        // ===========================================
        // STEP 350: MagnScanNGProcess
        // ===========================================
        STEP_ST10_Flow15_FRobot_3_MagnScanNGProcess:
            // No actions in XML

            // Transition to next step: 699
            IF TRUE THEN  // Sequential transition - review XML for actual condition
                #State := STEP_ST10_Flow15_FRobot_3_OKPutProcessFinish;
            END_IF;

        // ===========================================
        // STEP 699: OKPutProcessFinish
        // ===========================================
        STEP_ST10_Flow15_FRobot_3_OKPutProcessFinish:
            // Action Qualifier=S
            // Token: #ioPM_Inface.ProcessComplete
            #ioPM_Inface.ProcessComplete := TRUE;
            // Action Qualifier=R
            // Token: #ioPM_Inface.ProcessStart
            #ioPM_Inface.ProcessStart := FALSE;

            // Transition to next step: 355
            IF TRUE THEN  // Sequential transition - review XML for actual condition
                #State := STEP_ST10_Flow15_FRobot_3_StartRobotScanRing;
            END_IF;

        // ===========================================
        // STEP 355: StartRobotScanRing
        // ===========================================
        STEP_ST10_Flow15_FRobot_3_StartRobotScanRing:
            // Action Qualifier=N
            // Token: "KukaRobot3_CtrlDB".sPLCtoROB.User.Cycle.DI261_ScanRingReq
            "KukaRobot3_CtrlDB".sPLCtoROB.User.Cycle.DI261_ScanRingReq;

            // Transition to next step: 549
            IF TRUE THEN  // Sequential transition - review XML for actual condition
                #State := STEP_ST10_Flow15_FRobot_3_PressShaftPutProcessFinish;
            END_IF;

        // ===========================================
        // STEP 549: PressShaftPutProcessFinish
        // ===========================================
        STEP_ST10_Flow15_FRobot_3_PressShaftPutProcessFinish:
            // Action Qualifier=S
            // Token: #ioPM_Inface.ProcessComplete
            #ioPM_Inface.ProcessComplete := TRUE;
            // Action Qualifier=R
            // Token: #ioPM_Inface.ProcessStart
            #ioPM_Inface.ProcessStart := FALSE;

            // Transition to next step: 255
            IF TRUE THEN  // Sequential transition - review XML for actual condition
                #State := STEP_ST10_Flow15_FRobot_3_DataMove_1;
            END_IF;

        // ===========================================
        // STEP 255: DataMove_1
        // ===========================================
        STEP_ST10_Flow15_FRobot_3_DataMove_1:
            // Action Qualifier=N, Event="S1"
            // Token: "AutoProcessData".F_Robot3Grip2 := "AutoProcessData".C_MagnScanNGBuffer
            "AutoProcessData".F_Robot3Grip2 := "AutoProcessData".C_MagnScanNGBuffer;
            // Action Qualifier=N, Event="S1"
            // Token: "AutoProcessData".C_MagnScanNGBuffer := "AutoProcessData".ClearData
            "AutoProcessData".C_MagnScanNGBuffer := "AutoProcessData".ClearData;

            // Transition to next step: 382
            IF TRUE THEN  // Sequential transition - review XML for actual condition
                #State := STEP_ST10_Flow15_FRobot_3_Grip2SensorError;
            END_IF;

        // ===========================================
        // STEP 382: Grip2SensorError
        // ===========================================
        STEP_ST10_Flow15_FRobot_3_Grip2SensorError:
            // Action Qualifier=S
            // Token: "ST10_DeviceError".F.Robot_3.Grip2SensorCheckError
            "ST10_DeviceError".F.Robot_3.Grip2SensorCheckError := TRUE;

            // Transition to next step: 253
            IF TRUE THEN  // Sequential transition - review XML for actual condition
                #State := STEP_ST10_Flow15_FRobot_3_DataMove;
            END_IF;

        // ===========================================
        // STEP 253: DataMove
        // ===========================================
        STEP_ST10_Flow15_FRobot_3_DataMove:
            // Action Qualifier=N, Event="S1"
            // Token: "AutoProcessData".F_Robot3Grip1 := "AutoProcessData".C_GlueNGBuffer
            "AutoProcessData".F_Robot3Grip1 := "AutoProcessData".C_GlueNGBuffer;
            // Action Qualifier=N, Event="S1"
            // Token: "AutoProcessData".C_GlueNGBuffer := "AutoProcessData".ClearData
            "AutoProcessData".C_GlueNGBuffer := "AutoProcessData".ClearData;

            // Transition to next step: 919
            IF TRUE THEN  // Sequential transition - review XML for actual condition
                #State := STEP_ST10_Flow15_FRobot_3_MasteringTestFinish;
            END_IF;

        // ===========================================
        // STEP 919: MasteringTestFinish
        // ===========================================
        STEP_ST10_Flow15_FRobot_3_MasteringTestFinish:
            // Action Qualifier=R
            // Token: "Robot_DB".Robot_3.MasteringTest_Req
            "Robot_DB".Robot_3.MasteringTest_Req := FALSE;

            // Transition to next step: 900
            IF TRUE THEN  // Sequential transition - review XML for actual condition
                #State := STEP_ST10_Flow15_FRobot_3_S_900;
            END_IF;

        // ===========================================
        // STEP 900: 900
        // ===========================================
        STEP_ST10_Flow15_FRobot_3_S_900:
            // No actions in XML

            // Transition to next step: 309
            IF TRUE THEN  // Sequential transition - review XML for actual condition
                #State := STEP_ST10_Flow15_FRobot_3_WaitRobotReachPos1;
            END_IF;

        // ===========================================
        // STEP 309: WaitRobotReachPos1
        // ===========================================
        STEP_ST10_Flow15_FRobot_3_WaitRobotReachPos1:
            // No actions in XML

            // Transition to next step: 335
            IF TRUE THEN  // Sequential transition - review XML for actual condition
                #State := STEP_ST10_Flow15_FRobot_3_RobotScanGripperReachPos1;
            END_IF;

        // ===========================================
        // STEP 335: RobotScanGripperReachPos1
        // ===========================================
        STEP_ST10_Flow15_FRobot_3_RobotScanGripperReachPos1:
            // No actions in XML

            // Transition to next step: 267
            IF TRUE THEN  // Sequential transition - review XML for actual condition
                #State := STEP_ST10_Flow15_FRobot_3_Data_Clear_7;
            END_IF;

        // ===========================================
        // STEP 267: Data Clear_7
        // ===========================================
        STEP_ST10_Flow15_FRobot_3_Data_Clear_7:
            // Action Qualifier=N, Event="S1"
            // Token: "AutoProcessData".F_Robot3Grip1 := "AutoProcessData".ClearData
            "AutoProcessData".F_Robot3Grip1 := "AutoProcessData".ClearData;

            // Transition to next step: 705
            IF TRUE THEN  // Sequential transition - review XML for actual condition
                #State := STEP_ST10_Flow15_FRobot_3_WaitR1MaintenPosFinsh_1;
            END_IF;

        // ===========================================
        // STEP 705: WaitR1MaintenPosFinsh_1
        // ===========================================
        STEP_ST10_Flow15_FRobot_3_WaitR1MaintenPosFinsh_1:
            // Action Qualifier=R
            // Token: "AutoProcessControl".Robot_3.MaintenanceRequest
            "AutoProcessControl".Robot_3.MaintenanceRequest := FALSE;

            // Transition to next step: 500
            IF TRUE THEN  // Sequential transition - review XML for actual condition
                #State := STEP_ST10_Flow15_FRobot_3_PressShaftPutProcess;
            END_IF;

        // ===========================================
        // STEP 500: PressShaftPutProcess
        // ===========================================
        STEP_ST10_Flow15_FRobot_3_PressShaftPutProcess:
            // No actions in XML

            // Transition to next step: 376
            IF TRUE THEN  // Sequential transition - review XML for actual condition
                #State := STEP_ST10_Flow15_FRobot_3_StartRobotNG3Put;
            END_IF;

        // ===========================================
        // STEP 376: StartRobotNG3Put
        // ===========================================
        STEP_ST10_Flow15_FRobot_3_StartRobotNG3Put:
            // Action Qualifier=N
            // Token: "KukaRobot3_CtrlDB".sPLCtoROB.User.Cycle.DI267_LoadScanNGReq3
            "KukaRobot3_CtrlDB".sPLCtoROB.User.Cycle.DI267_LoadScanNGReq3;

            // Transition to next step: 333
            IF TRUE THEN  // Sequential transition - review XML for actual condition
                #State := STEP_ST10_Flow15_FRobot_3_RobotTaskSelect;
            END_IF;

        // ===========================================
        // STEP 333: RobotTaskSelect
        // ===========================================
        STEP_ST10_Flow15_FRobot_3_RobotTaskSelect:
            // No actions in XML

            // Transition to next step: 800
            IF TRUE THEN  // Sequential transition - review XML for actual condition
                #State := STEP_ST10_Flow15_FRobot_3_NG_3_PutProcess;
            END_IF;

        // ===========================================
        // STEP 800: NG 3 PutProcess
        // ===========================================
        STEP_ST10_Flow15_FRobot_3_NG_3_PutProcess:
            // No actions in XML

            // Transition to next step: 133
            IF TRUE THEN  // Sequential transition - review XML for actual condition
                #State := STEP_ST10_Flow15_FRobot_3_Brake_Test;
            END_IF;

        // ===========================================
        // STEP 133: Brake_Test
        // ===========================================
        STEP_ST10_Flow15_FRobot_3_Brake_Test:
            // Action Qualifier=R
            // Token: #ioPM_Inface.ProcessComplete
            #ioPM_Inface.ProcessComplete := FALSE;
            // Action Qualifier=S
            // Token: #ioPM_Inface.ProcessStart
            #ioPM_Inface.ProcessStart := TRUE;

            // Transition to next step: 365
            IF TRUE THEN  // Sequential transition - review XML for actual condition
                #State := STEP_ST10_Flow15_FRobot_3_WaitRobotFinish_7;
            END_IF;

        // ===========================================
        // STEP 365: WaitRobotFinish_7
        // ===========================================
        STEP_ST10_Flow15_FRobot_3_WaitRobotFinish_7:
            // No actions in XML

            // Transition to next step: 331
            IF TRUE THEN  // Sequential transition - review XML for actual condition
                #State := STEP_ST10_Flow15_FRobot_3_Gripe1StatusAlarm;
            END_IF;

        // ===========================================
        // STEP 331: Gripe1StatusAlarm
        // ===========================================
        STEP_ST10_Flow15_FRobot_3_Gripe1StatusAlarm:
            // Action Qualifier=S
            // Token: "ST10_DeviceError".F.Robot_3.Grip1Error
            "ST10_DeviceError".F.Robot_3.Grip1Error := TRUE;

            // Transition to next step: 372
            IF TRUE THEN  // Sequential transition - review XML for actual condition
                #State := STEP_ST10_Flow15_FRobot_3_WaitRobotGripStatus_4;
            END_IF;

        // ===========================================
        // STEP 372: WaitRobotGripStatus_4
        // ===========================================
        STEP_ST10_Flow15_FRobot_3_WaitRobotGripStatus_4:
            // No actions in XML

            // Transition to next step: 265
            IF TRUE THEN  // Sequential transition - review XML for actual condition
                #State := STEP_ST10_Flow15_FRobot_3_Data_Clear_6;
            END_IF;

        // ===========================================
        // STEP 265: Data Clear_6
        // ===========================================
        STEP_ST10_Flow15_FRobot_3_Data_Clear_6:
            // Action Qualifier=N
            // Token: "Robot_DB".Robot_3.SpeedCount := "Robot_DB".Robot_3.SpeedCount + 1
            "Robot_DB".Robot_3.SpeedCount := "Robot_DB".Robot_3.SpeedCount + 1;

            // Transition to next step: 2
            IF TRUE THEN  // Sequential transition - review XML for actual condition
                #State := STEP_ST10_Flow15_FRobot_3_S2;
            END_IF;

        // ===========================================
        // STEP 2: S2
        // ===========================================
        STEP_ST10_Flow15_FRobot_3_S2:
            // No actions in XML

            // Transition to next step: 245
            IF TRUE THEN  // Sequential transition - review XML for actual condition
                #State := STEP_ST10_Flow15_FRobot_3_CheckScanReady;
            END_IF;

        // ===========================================
        // STEP 245: CheckScanReady
        // ===========================================
        STEP_ST10_Flow15_FRobot_3_CheckScanReady:
            // No actions in XML

            // Transition to next step: 8
            IF TRUE THEN  // Sequential transition - review XML for actual condition
                #State := STEP_ST10_Flow15_FRobot_3_S8;
            END_IF;

        // ===========================================
        // STEP 8: S8
        // ===========================================
        STEP_ST10_Flow15_FRobot_3_S8:
            // No actions in XML

            // Transition to next step: 248
            IF TRUE THEN  // Sequential transition - review XML for actual condition
                #State := STEP_ST10_Flow15_FRobot_3_CodeMove;
            END_IF;

        // ===========================================
        // STEP 248: CodeMove
        // ===========================================
        STEP_ST10_Flow15_FRobot_3_CodeMove:
            // Action Qualifier=N
            // Token: "AutoProcessData".F_Robot3Grip2.RingCode_2 := "KeyenceSR1000Ctrl_803A1DB".sHMI.Status.CurrentCode
            "AutoProcessData".F_Robot3Grip2.RingCode_2 := "KeyenceSR1000Ctrl_803A1DB".sHMI.Status.CurrentCode;

            // Transition to next step: 347
            IF TRUE THEN  // Sequential transition - review XML for actual condition
                #State := STEP_ST10_Flow15_FRobot_3_WaitRobotGripHaveStatus_1;
            END_IF;

        // ===========================================
        // STEP 347: WaitRobotGripHaveStatus_1
        // ===========================================
        STEP_ST10_Flow15_FRobot_3_WaitRobotGripHaveStatus_1:
            // No actions in XML

    END_CASE;

    // UPDATE ioPM_Inface
    #ioPM_Inface.InitialRun := #act_InitialRun;
    #ioPM_Inface.InitialOK := #act_InitialOK;
    #ioPM_Inface.WaitRunning := #act_WaitRunning;
    #ioPM_Inface.Running := #act_Running;
    #ioPM_Inface.ProcessComplete := #act_ProcessComplete;
    #ioPM_Inface.ProcessStart := #act_ProcessStart;
    #ioPM_Inface.UnPause := #act_UnPause;

    // ERROR HANDLING
    IF #bError THEN
        #ioStatus := 900;
        #oAlarmID := INT_TO_WORD(#wErrorID);
    ELSE
        #ioStatus := 0;
        #oAlarmID := 0;
    END_IF;
END_FUNCTION_BLOCK

//=============================================================================
// END OF FILE
//=============================================================================
